PROGRAM MAIN
VAR
	fHysteresis: REAL := 1;
	fbSR: SR;
END_VAR
VAR // added by the converter: edge detectors and wires of the graphical bodies
    _w1, _w2 : ANY;
END_VAR

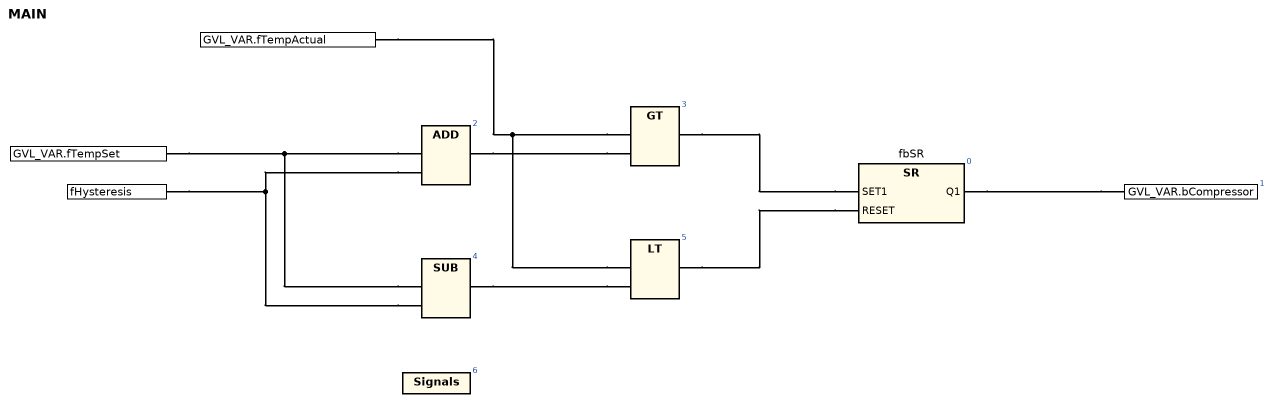
fbSR(SET1 := _w1, RESET := _w2); // SR
GVL_VAR.bCompressor := fbSR.Q1;
_w1 := GVL_VAR.fTempActual > GVL_VAR.fTempSet + fHysteresis;
_w2 := GVL_VAR.fTempActual < GVL_VAR.fTempSet - fHysteresis;
Signals();

END_PROGRAM

(* stored: Version 1.1.0.1, ProductVersion 3.1.4024.12
   POU MAIN: Id {d1ab3f02-411b-43c7-b8c2-7d6370a49feb}, SpecialFunc None *)
